FUNCTION_BLOCK CfbOvercurrentDetector
  (* Standard: 61499-2 *)
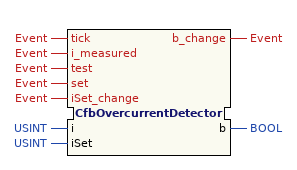
  EVENT_INPUT
    tick;
    i_measured;
    test;
    set;
    iSet_change;
  END_EVENT
  EVENT_OUTPUT
    b_change;
  END_EVENT
  VAR_INPUT
    i : USINT;
    iSet : USINT;
  END_VAR
  VAR_OUTPUT
    b : BOOL;
  END_VAR
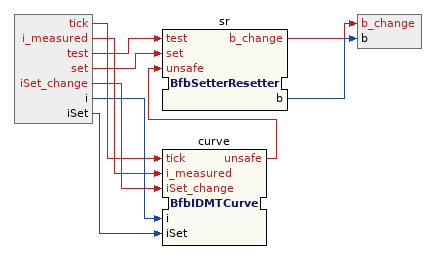
  FBS
    sr : BfbSetterResetter;
    curve : BfbIDMTCurve;
  END_FBS
  EVENT_CONNECTIONS
    tick TO curve.tick;
    i_measured TO curve.i_measured;
    iSet_change TO curve.iSet_change;
    test TO sr.test;
    set TO sr.set;
    curve.unsafe TO sr.unsafe;
    sr.b_change TO b_change;
  END_CONNECTIONS
  DATA_CONNECTIONS
    i TO curve.i;
    iSet TO curve.iSet;
    sr.b TO b;
  END_CONNECTIONS
END_FUNCTION_BLOCK
